// TIA Portal V17 export
// export: Created 2023-02-13T11:16:24.8420707Z, ExportSetting WithDefaults, DisplayName Totally Integrated Automation Portal, DisplayVersion V17, DisplayName TIA Portal Openness, DisplayVersion V17, DisplayName TIA Portal Teamcenter Gateway, DisplayVersion V17, DisplayName TIA Portal Version Control Interface, DisplayVersion V17, DisplayName SINAMICS Startdrive Advanced, DisplayVersion V17, DisplayName SINAMICS Startdrive G130, G150, S120, S150, SINAMICS MV, S210, DisplayVersion V17, DisplayName SINAMICS Startdrive G110M, G120, G120C, G120D, G120P, G115D, DisplayVersion V17, DisplayName STEP 7 Professional, DisplayVersion V17, DisplayName STEP 7 Safety, DisplayVersion V17, DisplayName WinCC Professional, DisplayVersion V17
FUNCTION_BLOCK "IO Analog Storage"   // FB11, LAD
{ S7_Optimized_Access := 'FALSE' }
VERSION : 0.1
// stored: AutoNumber true, IsIECCheckEnabled false, SetENOAutomatically false, UDAEnableTagReadback false
   VAR_INPUT
      Init : Bool;
      Reset : Bool;
   END_VAR
   VAR
      "LT-23.01" : "Ana_w_K1K2";
      "LT-24.01" : "Ana_w_K1K2";
      "LT-33.01" : "Ana_w_K1K2";
      "LT-34.01" { S7_SetPoint := 'True'} : "Ana_w_K1K2";
      "LT-35.01" { S7_SetPoint := 'True'} : "Ana_w_K1K2";
      "LT-79.01" { S7_SetPoint := 'True'} : "Ana_w_K1K2";
      "LT-81.01" { S7_SetPoint := 'True'} : "Ana_w_K1K2";
      "LT-84.01" { S7_SetPoint := 'True'} : "Ana_w_K1K2";
      "LT-82.01" { S7_SetPoint := 'True'} : "Ana_w_K1K2";
   END_VAR
BEGIN

REGION Network 1: LT-23.01
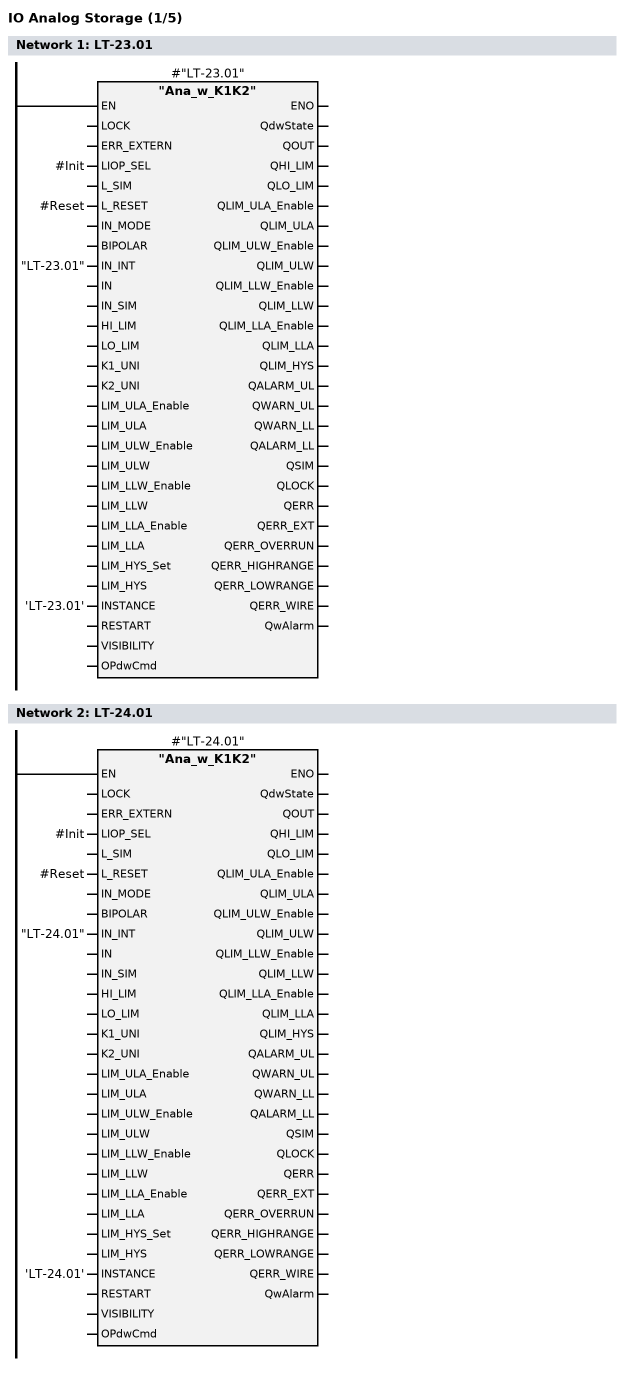
   RUNG wire#powerrail
      #"LT-23.01"(LOCK :=, ERR_EXTERN :=, LIOP_SEL := #Init, L_SIM :=, L_RESET := #Reset, IN_MODE :=, BIPOLAR :=, IN_INT := "LT-23.01", IN :=, IN_SIM :=, HI_LIM :=, LO_LIM :=, K1_UNI :=, K2_UNI :=, LIM_ULA_Enable :=, LIM_ULA :=, LIM_ULW_Enable :=, LIM_ULW :=, LIM_LLW_Enable :=, LIM_LLW :=, LIM_LLA_Enable :=, LIM_LLA :=, LIM_HYS_Set :=, LIM_HYS :=, INSTANCE := 'LT-23.01', RESTART :=, VISIBILITY :=, OPdwCmd :=, QdwState =>, QOUT =>, QHI_LIM =>, QLO_LIM =>, QLIM_ULA_Enable =>, QLIM_ULA =>, QLIM_ULW_Enable =>, QLIM_ULW =>, QLIM_LLW_Enable =>, QLIM_LLW =>, QLIM_LLA_Enable =>, QLIM_LLA =>, QLIM_HYS =>, QALARM_UL =>, QWARN_UL =>, QWARN_LL =>, QALARM_LL =>, QSIM =>, QLOCK =>, QERR =>, QERR_EXT =>, QERR_OVERRUN =>, QERR_HIGHRANGE =>, QERR_LOWRANGE =>, QERR_WIRE =>, QwAlarm =>)
   END_RUNG
   // the same network as SCL:
   #"LT-23.01"(LIOP_SEL := #Init, L_RESET := #Reset, IN_INT := "LT-23.01", INSTANCE := 'LT-23.01');   // "Ana_w_K1K2"
END_REGION

REGION Network 2: LT-24.01
   RUNG wire#powerrail
      #"LT-24.01"(LOCK :=, ERR_EXTERN :=, LIOP_SEL := #Init, L_SIM :=, L_RESET := #Reset, IN_MODE :=, BIPOLAR :=, IN_INT := "LT-24.01", IN :=, IN_SIM :=, HI_LIM :=, LO_LIM :=, K1_UNI :=, K2_UNI :=, LIM_ULA_Enable :=, LIM_ULA :=, LIM_ULW_Enable :=, LIM_ULW :=, LIM_LLW_Enable :=, LIM_LLW :=, LIM_LLA_Enable :=, LIM_LLA :=, LIM_HYS_Set :=, LIM_HYS :=, INSTANCE := 'LT-24.01', RESTART :=, VISIBILITY :=, OPdwCmd :=, QdwState =>, QOUT =>, QHI_LIM =>, QLO_LIM =>, QLIM_ULA_Enable =>, QLIM_ULA =>, QLIM_ULW_Enable =>, QLIM_ULW =>, QLIM_LLW_Enable =>, QLIM_LLW =>, QLIM_LLA_Enable =>, QLIM_LLA =>, QLIM_HYS =>, QALARM_UL =>, QWARN_UL =>, QWARN_LL =>, QALARM_LL =>, QSIM =>, QLOCK =>, QERR =>, QERR_EXT =>, QERR_OVERRUN =>, QERR_HIGHRANGE =>, QERR_LOWRANGE =>, QERR_WIRE =>, QwAlarm =>)
   END_RUNG
   // the same network as SCL:
   #"LT-24.01"(LIOP_SEL := #Init, L_RESET := #Reset, IN_INT := "LT-24.01", INSTANCE := 'LT-24.01');   // "Ana_w_K1K2"
END_REGION

REGION Network 3: LT-33.01
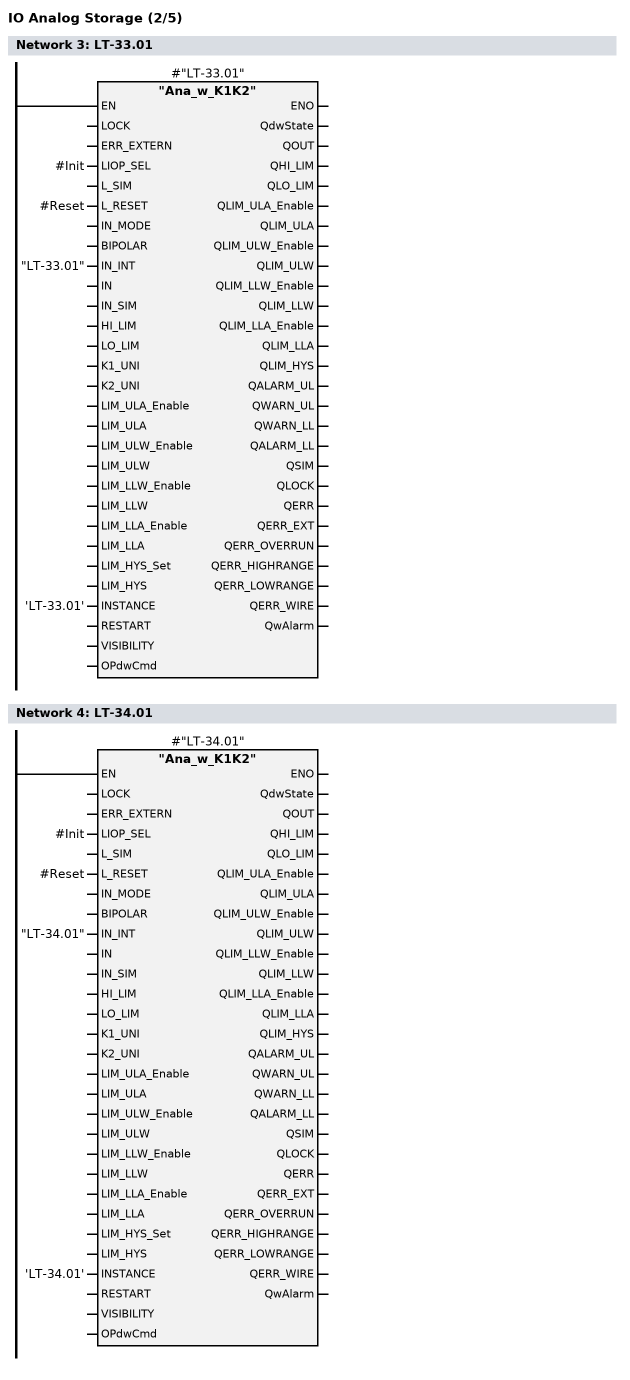
   RUNG wire#powerrail
      #"LT-33.01"(LOCK :=, ERR_EXTERN :=, LIOP_SEL := #Init, L_SIM :=, L_RESET := #Reset, IN_MODE :=, BIPOLAR :=, IN_INT := "LT-33.01", IN :=, IN_SIM :=, HI_LIM :=, LO_LIM :=, K1_UNI :=, K2_UNI :=, LIM_ULA_Enable :=, LIM_ULA :=, LIM_ULW_Enable :=, LIM_ULW :=, LIM_LLW_Enable :=, LIM_LLW :=, LIM_LLA_Enable :=, LIM_LLA :=, LIM_HYS_Set :=, LIM_HYS :=, INSTANCE := 'LT-33.01', RESTART :=, VISIBILITY :=, OPdwCmd :=, QdwState =>, QOUT =>, QHI_LIM =>, QLO_LIM =>, QLIM_ULA_Enable =>, QLIM_ULA =>, QLIM_ULW_Enable =>, QLIM_ULW =>, QLIM_LLW_Enable =>, QLIM_LLW =>, QLIM_LLA_Enable =>, QLIM_LLA =>, QLIM_HYS =>, QALARM_UL =>, QWARN_UL =>, QWARN_LL =>, QALARM_LL =>, QSIM =>, QLOCK =>, QERR =>, QERR_EXT =>, QERR_OVERRUN =>, QERR_HIGHRANGE =>, QERR_LOWRANGE =>, QERR_WIRE =>, QwAlarm =>)
   END_RUNG
   // the same network as SCL:
   #"LT-33.01"(LIOP_SEL := #Init, L_RESET := #Reset, IN_INT := "LT-33.01", INSTANCE := 'LT-33.01');   // "Ana_w_K1K2"
END_REGION

REGION Network 4: LT-34.01
   RUNG wire#powerrail
      #"LT-34.01"(LOCK :=, ERR_EXTERN :=, LIOP_SEL := #Init, L_SIM :=, L_RESET := #Reset, IN_MODE :=, BIPOLAR :=, IN_INT := "LT-34.01", IN :=, IN_SIM :=, HI_LIM :=, LO_LIM :=, K1_UNI :=, K2_UNI :=, LIM_ULA_Enable :=, LIM_ULA :=, LIM_ULW_Enable :=, LIM_ULW :=, LIM_LLW_Enable :=, LIM_LLW :=, LIM_LLA_Enable :=, LIM_LLA :=, LIM_HYS_Set :=, LIM_HYS :=, INSTANCE := 'LT-34.01', RESTART :=, VISIBILITY :=, OPdwCmd :=, QdwState =>, QOUT =>, QHI_LIM =>, QLO_LIM =>, QLIM_ULA_Enable =>, QLIM_ULA =>, QLIM_ULW_Enable =>, QLIM_ULW =>, QLIM_LLW_Enable =>, QLIM_LLW =>, QLIM_LLA_Enable =>, QLIM_LLA =>, QLIM_HYS =>, QALARM_UL =>, QWARN_UL =>, QWARN_LL =>, QALARM_LL =>, QSIM =>, QLOCK =>, QERR =>, QERR_EXT =>, QERR_OVERRUN =>, QERR_HIGHRANGE =>, QERR_LOWRANGE =>, QERR_WIRE =>, QwAlarm =>)
   END_RUNG
   // the same network as SCL:
   #"LT-34.01"(LIOP_SEL := #Init, L_RESET := #Reset, IN_INT := "LT-34.01", INSTANCE := 'LT-34.01');   // "Ana_w_K1K2"
END_REGION

REGION Network 5: LT-35.01
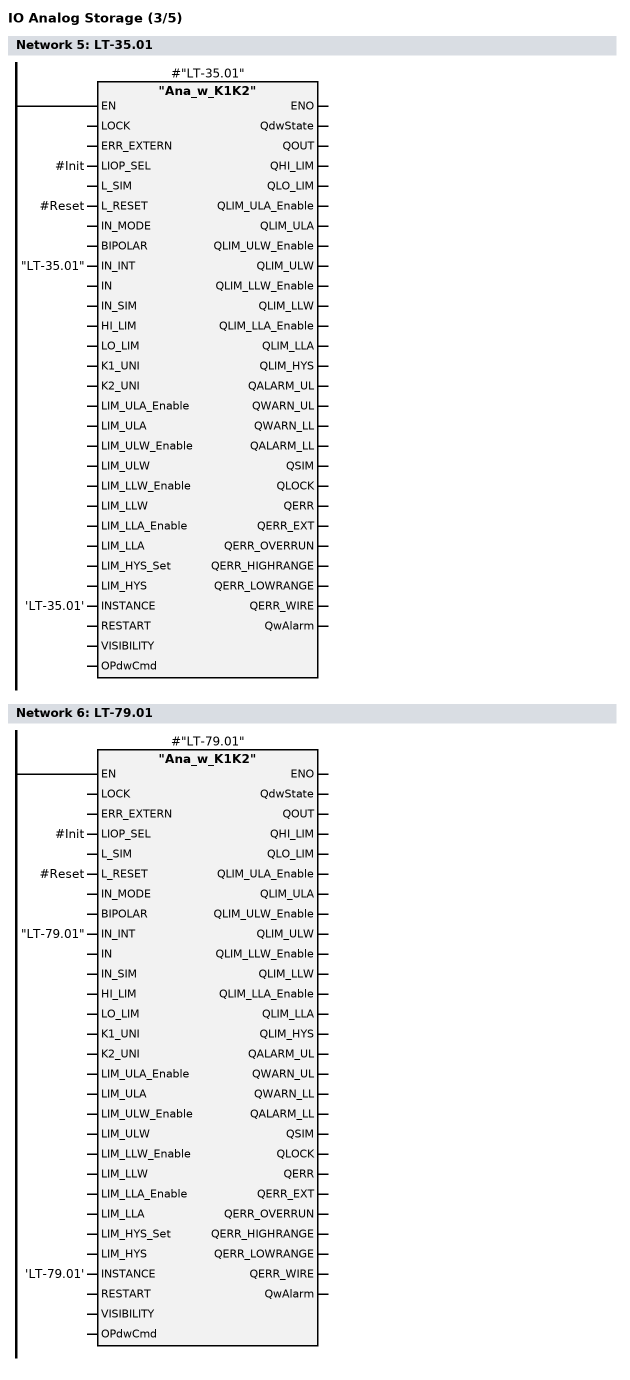
   RUNG wire#powerrail
      #"LT-35.01"(LOCK :=, ERR_EXTERN :=, LIOP_SEL := #Init, L_SIM :=, L_RESET := #Reset, IN_MODE :=, BIPOLAR :=, IN_INT := "LT-35.01", IN :=, IN_SIM :=, HI_LIM :=, LO_LIM :=, K1_UNI :=, K2_UNI :=, LIM_ULA_Enable :=, LIM_ULA :=, LIM_ULW_Enable :=, LIM_ULW :=, LIM_LLW_Enable :=, LIM_LLW :=, LIM_LLA_Enable :=, LIM_LLA :=, LIM_HYS_Set :=, LIM_HYS :=, INSTANCE := 'LT-35.01', RESTART :=, VISIBILITY :=, OPdwCmd :=, QdwState =>, QOUT =>, QHI_LIM =>, QLO_LIM =>, QLIM_ULA_Enable =>, QLIM_ULA =>, QLIM_ULW_Enable =>, QLIM_ULW =>, QLIM_LLW_Enable =>, QLIM_LLW =>, QLIM_LLA_Enable =>, QLIM_LLA =>, QLIM_HYS =>, QALARM_UL =>, QWARN_UL =>, QWARN_LL =>, QALARM_LL =>, QSIM =>, QLOCK =>, QERR =>, QERR_EXT =>, QERR_OVERRUN =>, QERR_HIGHRANGE =>, QERR_LOWRANGE =>, QERR_WIRE =>, QwAlarm =>)
   END_RUNG
   // the same network as SCL:
   #"LT-35.01"(LIOP_SEL := #Init, L_RESET := #Reset, IN_INT := "LT-35.01", INSTANCE := 'LT-35.01');   // "Ana_w_K1K2"
END_REGION

REGION Network 6: LT-79.01
   RUNG wire#powerrail
      #"LT-79.01"(LOCK :=, ERR_EXTERN :=, LIOP_SEL := #Init, L_SIM :=, L_RESET := #Reset, IN_MODE :=, BIPOLAR :=, IN_INT := "LT-79.01", IN :=, IN_SIM :=, HI_LIM :=, LO_LIM :=, K1_UNI :=, K2_UNI :=, LIM_ULA_Enable :=, LIM_ULA :=, LIM_ULW_Enable :=, LIM_ULW :=, LIM_LLW_Enable :=, LIM_LLW :=, LIM_LLA_Enable :=, LIM_LLA :=, LIM_HYS_Set :=, LIM_HYS :=, INSTANCE := 'LT-79.01', RESTART :=, VISIBILITY :=, OPdwCmd :=, QdwState =>, QOUT =>, QHI_LIM =>, QLO_LIM =>, QLIM_ULA_Enable =>, QLIM_ULA =>, QLIM_ULW_Enable =>, QLIM_ULW =>, QLIM_LLW_Enable =>, QLIM_LLW =>, QLIM_LLA_Enable =>, QLIM_LLA =>, QLIM_HYS =>, QALARM_UL =>, QWARN_UL =>, QWARN_LL =>, QALARM_LL =>, QSIM =>, QLOCK =>, QERR =>, QERR_EXT =>, QERR_OVERRUN =>, QERR_HIGHRANGE =>, QERR_LOWRANGE =>, QERR_WIRE =>, QwAlarm =>)
   END_RUNG
   // the same network as SCL:
   #"LT-79.01"(LIOP_SEL := #Init, L_RESET := #Reset, IN_INT := "LT-79.01", INSTANCE := 'LT-79.01');   // "Ana_w_K1K2"
END_REGION

REGION Network 7: LT-81.01
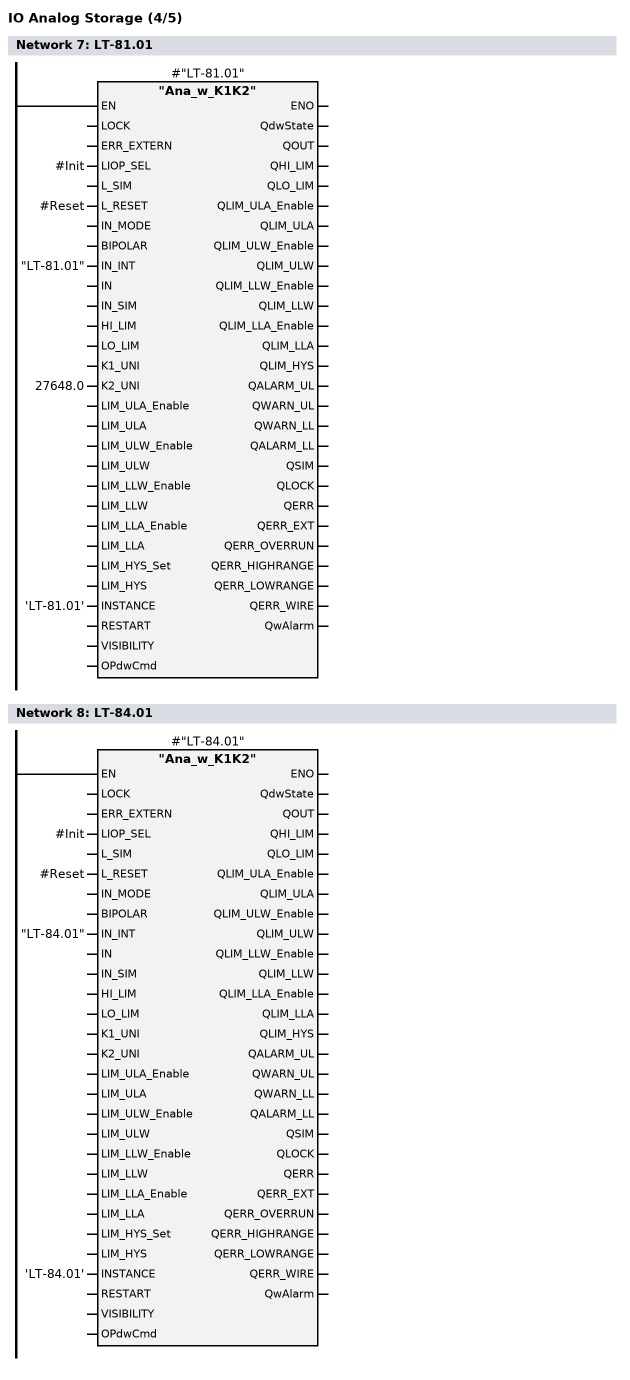
   RUNG wire#powerrail
      #"LT-81.01"(LOCK :=, ERR_EXTERN :=, LIOP_SEL := #Init, L_SIM :=, L_RESET := #Reset, IN_MODE :=, BIPOLAR :=, IN_INT := "LT-81.01", IN :=, IN_SIM :=, HI_LIM :=, LO_LIM :=, K1_UNI :=, K2_UNI := 27648.0, LIM_ULA_Enable :=, LIM_ULA :=, LIM_ULW_Enable :=, LIM_ULW :=, LIM_LLW_Enable :=, LIM_LLW :=, LIM_LLA_Enable :=, LIM_LLA :=, LIM_HYS_Set :=, LIM_HYS :=, INSTANCE := 'LT-81.01', RESTART :=, VISIBILITY :=, OPdwCmd :=, QdwState =>, QOUT =>, QHI_LIM =>, QLO_LIM =>, QLIM_ULA_Enable =>, QLIM_ULA =>, QLIM_ULW_Enable =>, QLIM_ULW =>, QLIM_LLW_Enable =>, QLIM_LLW =>, QLIM_LLA_Enable =>, QLIM_LLA =>, QLIM_HYS =>, QALARM_UL =>, QWARN_UL =>, QWARN_LL =>, QALARM_LL =>, QSIM =>, QLOCK =>, QERR =>, QERR_EXT =>, QERR_OVERRUN =>, QERR_HIGHRANGE =>, QERR_LOWRANGE =>, QERR_WIRE =>, QwAlarm =>)
   END_RUNG
   // the same network as SCL:
   #"LT-81.01"(LIOP_SEL := #Init,   // "Ana_w_K1K2"
               L_RESET := #Reset,
               IN_INT := "LT-81.01",
               K2_UNI := 27648.0,
               INSTANCE := 'LT-81.01');
END_REGION

REGION Network 8: LT-84.01
   RUNG wire#powerrail
      #"LT-84.01"(LOCK :=, ERR_EXTERN :=, LIOP_SEL := #Init, L_SIM :=, L_RESET := #Reset, IN_MODE :=, BIPOLAR :=, IN_INT := "LT-84.01", IN :=, IN_SIM :=, HI_LIM :=, LO_LIM :=, K1_UNI :=, K2_UNI :=, LIM_ULA_Enable :=, LIM_ULA :=, LIM_ULW_Enable :=, LIM_ULW :=, LIM_LLW_Enable :=, LIM_LLW :=, LIM_LLA_Enable :=, LIM_LLA :=, LIM_HYS_Set :=, LIM_HYS :=, INSTANCE := 'LT-84.01', RESTART :=, VISIBILITY :=, OPdwCmd :=, QdwState =>, QOUT =>, QHI_LIM =>, QLO_LIM =>, QLIM_ULA_Enable =>, QLIM_ULA =>, QLIM_ULW_Enable =>, QLIM_ULW =>, QLIM_LLW_Enable =>, QLIM_LLW =>, QLIM_LLA_Enable =>, QLIM_LLA =>, QLIM_HYS =>, QALARM_UL =>, QWARN_UL =>, QWARN_LL =>, QALARM_LL =>, QSIM =>, QLOCK =>, QERR =>, QERR_EXT =>, QERR_OVERRUN =>, QERR_HIGHRANGE =>, QERR_LOWRANGE =>, QERR_WIRE =>, QwAlarm =>)
   END_RUNG
   // the same network as SCL:
   #"LT-84.01"(LIOP_SEL := #Init, L_RESET := #Reset, IN_INT := "LT-84.01", INSTANCE := 'LT-84.01');   // "Ana_w_K1K2"
END_REGION

REGION Network 9: LT-82.01
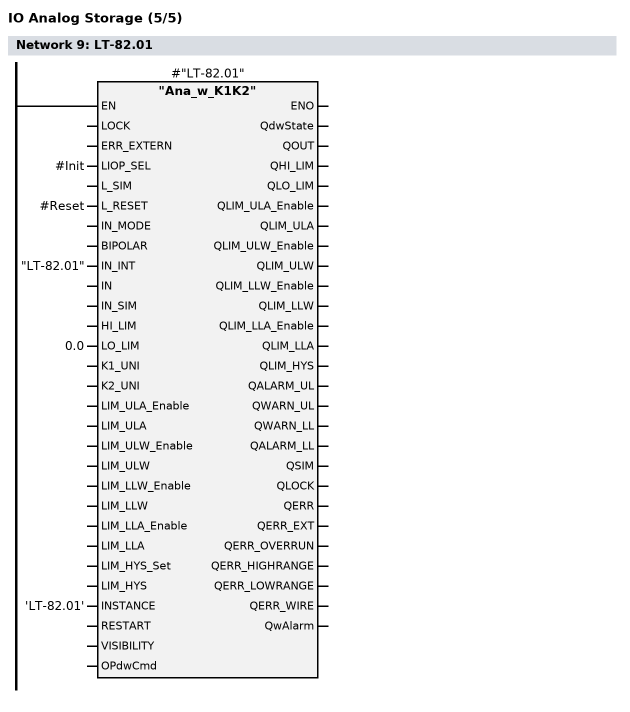
   RUNG wire#powerrail
      #"LT-82.01"(LOCK :=, ERR_EXTERN :=, LIOP_SEL := #Init, L_SIM :=, L_RESET := #Reset, IN_MODE :=, BIPOLAR :=, IN_INT := "LT-82.01", IN :=, IN_SIM :=, HI_LIM :=, LO_LIM := 0.0, K1_UNI :=, K2_UNI :=, LIM_ULA_Enable :=, LIM_ULA :=, LIM_ULW_Enable :=, LIM_ULW :=, LIM_LLW_Enable :=, LIM_LLW :=, LIM_LLA_Enable :=, LIM_LLA :=, LIM_HYS_Set :=, LIM_HYS :=, INSTANCE := 'LT-82.01', RESTART :=, VISIBILITY :=, OPdwCmd :=, QdwState =>, QOUT =>, QHI_LIM =>, QLO_LIM =>, QLIM_ULA_Enable =>, QLIM_ULA =>, QLIM_ULW_Enable =>, QLIM_ULW =>, QLIM_LLW_Enable =>, QLIM_LLW =>, QLIM_LLA_Enable =>, QLIM_LLA =>, QLIM_HYS =>, QALARM_UL =>, QWARN_UL =>, QWARN_LL =>, QALARM_LL =>, QSIM =>, QLOCK =>, QERR =>, QERR_EXT =>, QERR_OVERRUN =>, QERR_HIGHRANGE =>, QERR_LOWRANGE =>, QERR_WIRE =>, QwAlarm =>)
   END_RUNG
   // the same network as SCL:
   #"LT-82.01"(LIOP_SEL := #Init,   // "Ana_w_K1K2"
               L_RESET := #Reset,
               IN_INT := "LT-82.01",
               LO_LIM := 0.0,
               INSTANCE := 'LT-82.01');
END_REGION
END_FUNCTION_BLOCK
